TYPE ST_TestBasicControl_sub1 :
STRUCT
	sub1val	: DINT;
END_STRUCT
END_TYPE

(* stored: Version 1.1.0.1, ProductVersion 3.1.4024.9
   DUT ST_TestBasicControl_sub1: Id {b38d71a8-27b5-4641-9eec-6c3d505a108c} *)
